# EPICS autosave request: Db/NDFileHDF5XML_settings.req
$(P)$(R)TemplateFilePath
$(P)$(R)TemplateFileName
$(P)$(R)NDAttributesFile
$(P)$(R)EnableCallbacks
$(P)$(R)BlockingCallbacks
$(P)$(R)FileTemplate
$(P)$(R)FileWriteMode
$(P)$(R)FileName
$(P)$(R)FilePath
$(P)$(R)AutoSave
